Yaskawa INFORM job: REF_ODWLOK_NEW_X4.JBI

/JOB
//NAME REF_ODWLOK_NEW_X4
///FOLDERNAME INNE
//POS
///NPOS 13,13,0,0,0,0
///TOOL 0
///POSTYPE PULSE
///PULSE
C00000=28862,232315,242093,-120602,-126258,-18287
C00001=-85879,-96353,-67507,26769,-8866,29155
C00002=-90682,-94952,-60903,2018,-11322,40048
C00003=-108098,-110399,-80759,-62152,-14175,68196
C00004=-113513,-107421,-73683,-61030,-18975,67386
C00005=-107275,-157059,-86883,-25019,-29474,50696
C00006=-122154,-157663,-86910,-43091,-35033,57426
C00007=221370,-128165,-94668,86127,-52368,4397
C00008=222637,-115629,-85020,86703,-53233,4058
C00009=226166,-95549,-92179,97275,-55828,-4226
C00010=227012,-86748,-82897,96365,-56343,-3549
C00011=229160,-91044,-93793,98873,-58316,-5905
C00012=232489,-41307,-68674,103639,-62225,-10980
BC00000=270150,1327424,2
BC00001=7,705730,699321
BC00002=7,705730,699321
BC00003=7,705730,699321
BC00004=7,705730,699321
BC00005=4973,753652,1004101
BC00006=4973,753652,1004101
BC00007=188146,1353181,597486
BC00008=188146,1353181,597486
BC00009=188146,1353181,597486
BC00010=188146,1353181,597486
BC00011=208965,1347150,856546
BC00012=208965,1347150,856545
//INST
///DATE 2024/02/01 19:43
///ATTR SC,RW
///GROUP1 RB1,BS1
NOP
'FRONT
MOVJ C00000 BC00000 VJ=0.78 PL=0  //FRONT_RIGHT
'LEFT
MOVJ C00001 BC00001 VJ=0.78 PL=0  //1_SMALL
MOVJ C00002 BC00002 VJ=0.78 PL=0  //2_SMALL
MOVJ C00003 BC00003 VJ=0.78 PL=0  //3_SMALL
MOVJ C00004 BC00004 VJ=0.78 PL=0  //4_SMALL
MOVJ C00005 BC00005 VJ=0.78 PL=0  //1_LARGE
MOVJ C00006 BC00006 VJ=0.78 PL=0  //2_LARGE
'RIGHT
MOVJ C00007 BC00007 VJ=0.78 PL=0  //1_SMALL
MOVJ C00008 BC00008 VJ=0.78 PL=0  //2_SMALL
MOVJ C00009 BC00009 VJ=0.78 PL=0  //3_SMALL
MOVJ C00010 BC00010 VJ=0.78 PL=0  //4_SMALL
MOVJ C00011 BC00011 VJ=0.78 PL=0  //1_LARGE
MOVJ C00012 BC00012 VJ=0.78 PL=0  //2_LARGE
END
